// TIA Portal project "lab-3" (V12)

(* hardware
DEVICE "S7-1200 station_1"  SIMATIC 1200-Station
   slot 0: "S7-1200 rack"  Rack  V1.0
   slot 1: "PLC_1"  CPU 1214C AC/DC/Rly  6ES7 214-1BG31-0XB0  V3.0
      slot 3: "AQ1 x 12 bits_1"  6ES7 232-4HA30-0XB0  V1.0
*)

// ===== PLC "PLC_1"  CPU 1214C AC/DC/Rly =====

VAR_GLOBAL   // PLC tag table "Default tag table"
   "A" AT %M0.0 : Bool;
   "B" AT %M0.1 : Bool;
   "STOP" AT %I0.1 : Bool;
   "START" AT %I0.0 : Bool;
   "START-LATCH" AT %M0.2 : Bool;
   "C" AT %M0.3 : Bool;
   "TAG" AT %Q0.3 : Bool;
   "TAY" AT %Q0.4 : Bool;
   "TAR" AT %Q0.5 : Bool;
   "TBG" AT %Q0.0 : Bool;
   "TBY" AT %Q0.1 : Bool;
   "TBR" AT %Q0.2 : Bool;
   "PAG" AT %Q0.6 : Bool;
   "PAR" AT %Q0.7 : Bool;
   "PBG" AT %Q1.0 : Bool;
   "PBR" AT %Q1.1 : Bool;
   "S0" AT %M2.0 : Bool;
   "S1" AT %M2.1 : Bool;
   "S2" AT %M2.2 : Bool;
   "S3" AT %M2.3 : Bool;
   "S4" AT %M2.4 : Bool;
   "S4I" AT %M2.5 : Bool;
   "ba" AT %I0.2 : Bool;
   "bb" AT %I0.3 : Bool;
END_VAR

// folder: System blocks/Program resources

DATA_BLOCK "Tl"   // DB5
{ S7_Optimized_Access := 'FALSE' }
AUTHOR : Simatic
FAMILY : IEC
NAME : IEC_TMR
VERSION : 1.0
// stored: InstanceOfName ?
"?"
BEGIN
END_DATA_BLOCK

DATA_BLOCK "Ts"   // DB6
{ S7_Optimized_Access := 'FALSE' }
AUTHOR : Simatic
FAMILY : IEC
NAME : IEC_TMR
VERSION : 1.0
// stored: InstanceOfName ?
"?"
BEGIN
END_DATA_BLOCK

// folder: (top level)

ORGANIZATION_BLOCK "Main"   // OB1, LAD, ProgramCycle
TITLE = "Main Program Sweep (Cycle)"
{ S7_Optimized_Access := 'FALSE' }
VERSION : 0.1
BEGIN
END_ORGANIZATION_BLOCK